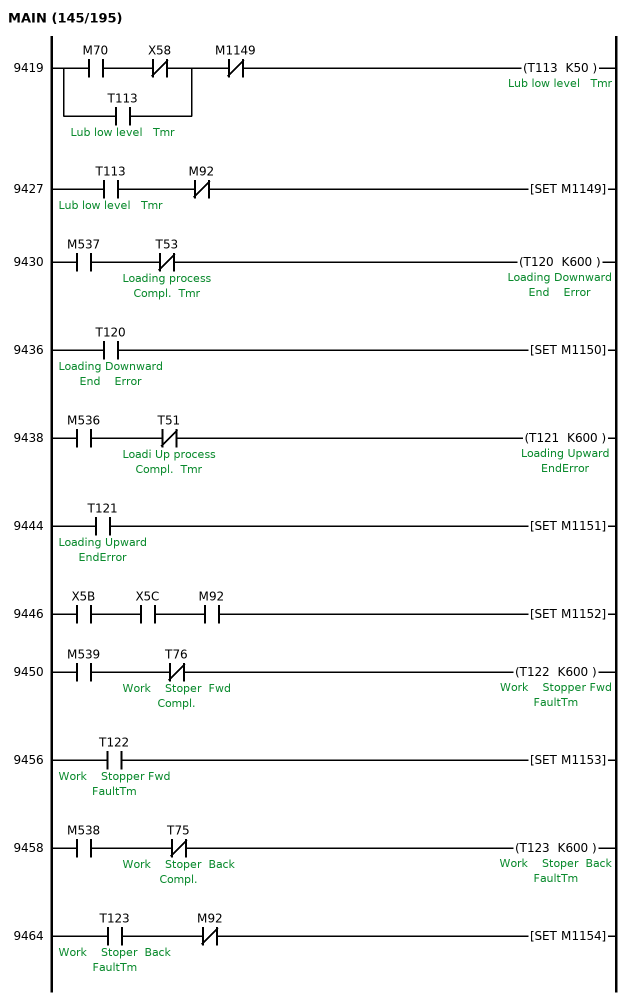
[picture p144: ladder of MAIN, rungs at steps 9419 to 9464]
9419  LD      M70
      ANI     X58
      OR      T113  ; Lub low level   Tmr
      ANI     M1149
      OUT     T113 K50  ; Lub low level   Tmr
9427  LD      T113  ; Lub low level   Tmr
      ANI     M92
      SET     M1149
9430  LD      M537
      ANI     T53  ; Loading process Compl.  Tmr
      OUT     T120 K600  ; Loading Downward End    Error
9436  LD      T120  ; Loading Downward End    Error
      SET     M1150
9438  LD      M536
      ANI     T51  ; Loadi Up process Compl.  Tmr
      OUT     T121 K600  ; Loading Upward  EndError
9444  LD      T121  ; Loading Upward  EndError
      SET     M1151
9446  LD      X5B
      AND     X5C
      AND     M92
      SET     M1152
9450  LD      M539
      ANI     T76  ; Work    Stoper  Fwd     Compl.
      OUT     T122 K600  ; Work    Stopper Fwd     FaultTm
9456  LD      T122  ; Work    Stopper Fwd     FaultTm
      SET     M1153
9458  LD      M538
      ANI     T75  ; Work    Stoper  Back    Compl.
      OUT     T123 K600  ; Work    Stoper  Back    FaultTm
9464  LD      T123  ; Work    Stoper  Back    FaultTm
      ANI     M92
      SET     M1154
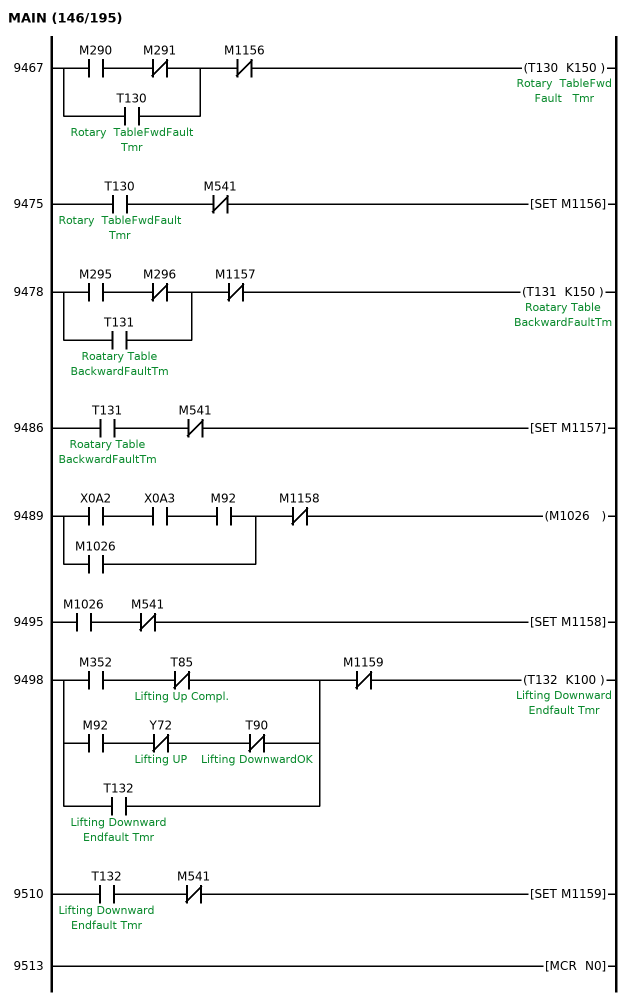
9467  LD      M290
      ANI     M291
      OR      T130  ; Rotary  TableFwdFault   Tmr
      ANI     M1156
      OUT     T130 K150  ; Rotary  TableFwdFault   Tmr
9475  LD      T130  ; Rotary  TableFwdFault   Tmr
      ANI     M541
      SET     M1156
9478  LD      M295
      ANI     M296
      OR      T131  ; Roatary Table   BackwardFaultTm
      ANI     M1157
      OUT     T131 K150  ; Roatary Table   BackwardFaultTm
9486  LD      T131  ; Roatary Table   BackwardFaultTm
      ANI     M541
      SET     M1157
9489  LD      X0A2
      AND     X0A3
      AND     M92
      OR      M1026
      ANI     M1158
      OUT     M1026
9495  LD      M1026
      ANI     M541
      SET     M1158
9498  LD      M352
      ANI     T85  ; Lifting Up Compl.
      LD      M92
      ANI     Y72  ; Lifting UP
      ANI     T90  ; Lifting DownwardOK
      ORB
      OR      T132  ; Lifting DownwardEndfault Tmr
      ANI     M1159
      OUT     T132 K100  ; Lifting DownwardEndfault Tmr
9510  LD      T132  ; Lifting DownwardEndfault Tmr
      ANI     M541
      SET     M1159
9513  MCR     N0
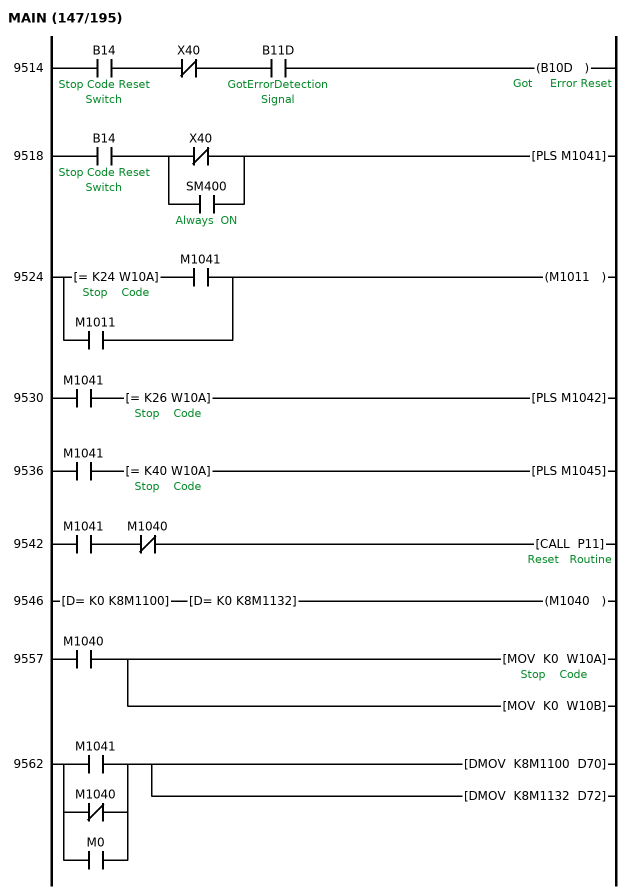
9514  LD      B14  ; Stop Code Reset Switch
      ANI     X40
      AND     B11D  ; GotErrorDetection Signal
      OUT     B10D  ; Got     Error Reset
9518  LD      B14  ; Stop Code Reset Switch
      LDI     X40
      OR      SM400  ; Always  ON
      ANB
      PLS     M1041
9524  LD=     K24 W10A  ; Stop    Code
      AND     M1041
      OR      M1011
      OUT     M1011
9530  LD      M1041
      AND=    K26 W10A  ; Stop    Code
      PLS     M1042
9536  LD      M1041
      AND=    K40 W10A  ; Stop    Code
      PLS     M1045
9542  LD      M1041
      ANI     M1040
      CALL    P11  ; Reset   Routine
9546  LDD=    K0 K8M1100
      ANDD=   K0 K8M1132
      OUT     M1040
9557  LD      M1040
      MOV     K0 W10A
      MOV     K0 W10B
9562  LD      M1041
      ORI     M1040
      OR      M0
      DMOV    K8M1100 D70
      DMOV    K8M1132 D72
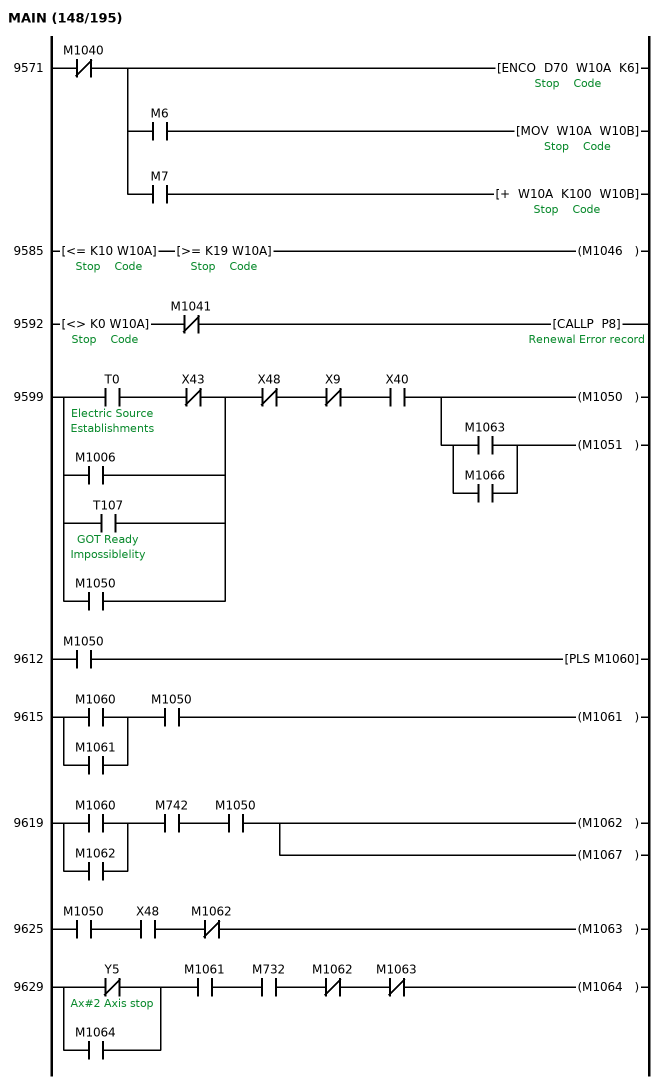
9571  LDI     M1040
      ENCO    D70 W10A K6
      MPS
      AND     M6
      MOV     W10A W10B
      MPP
      AND     M7
      +       W10A K100 W10B
9585  LD<=    K10 W10A  ; Stop    Code
      AND>=   K19 W10A  ; Stop    Code
      OUT     M1046
9592  LD<>    K0 W10A  ; Stop    Code
      ANI     M1041
      CALLP   P8  ; Renewal Error record
9599  LD      T0  ; Electric Source Establishments
      ANI     X43
      OR      M1006
      OR      T107  ; GOT Ready Impossiblelity
      OR      M1050
      ANI     X48
      ANI     X9
      AND     X40
      OUT     M1050
      LD      M1063
      OR      M1066
      ANB
      OUT     M1051
9612  LD      M1050
      PLS     M1060
9615  LD      M1060
      OR      M1061
      AND     M1050
      OUT     M1061
9619  LD      M1060
      OR      M1062
      AND     M742
      AND     M1050
      OUT     M1062
      OUT     M1067
9625  LD      M1050
      AND     X48
      ANI     M1062
      OUT     M1063
9629  LDI     Y5  ; Ax#2 Axis stop
      OR      M1064
      AND     M1061
      AND     M732
      ANI     M1062
      ANI     M1063
      OUT     M1064
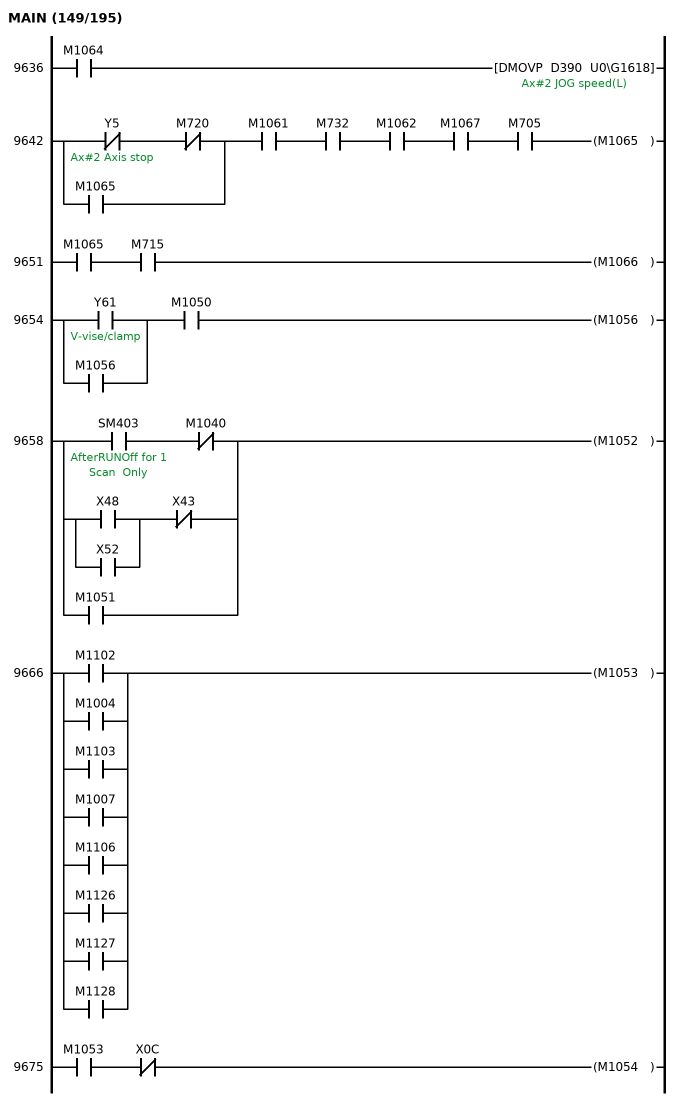
9636  LD      M1064
      DMOVP   D390 U0\G1618
9642  LDI     Y5  ; Ax#2 Axis stop
      ANI     M720
      OR      M1065
      AND     M1061
      AND     M732
      AND     M1062
      AND     M1067
      AND     M705
      OUT     M1065
9651  LD      M1065
      AND     M715
      OUT     M1066
9654  LD      Y61  ; V-vise/clamp
      OR      M1056
      AND     M1050
      OUT     M1056
9658  LD      SM403  ; AfterRUNOff for 1 Scan  Only
      ANI     M1040
      LD      X48
      OR      X52
      ANI     X43
      ORB
      OR      M1051
      OUT     M1052
9666  LD      M1102
      OR      M1004
      OR      M1103
      OR      M1007
      OR      M1106
      OR      M1126
      OR      M1127
      OR      M1128
      OUT     M1053
9675  LD      M1053
      ANI     X0C
      OUT     M1054
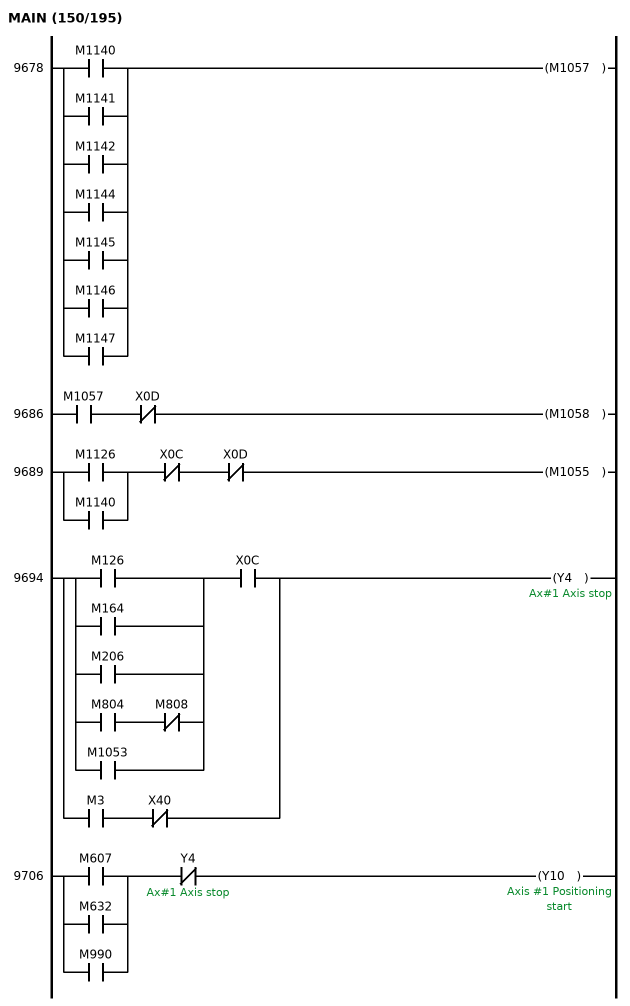
9678  LD      M1140
      OR      M1141
      OR      M1142
      OR      M1144
      OR      M1145
      OR      M1146
      OR      M1147
      OUT     M1057
9686  LD      M1057
      ANI     X0D
      OUT     M1058
9689  LD      M1126
      OR      M1140
      ANI     X0C
      ANI     X0D
      OUT     M1055
9694  LD      M126
      OR      M164
      OR      M206
      LD      M804
      ANI     M808
      ORB
      OR      M1053
      AND     X0C
      LD      M3
      ANI     X40
      ORB
      OUT     Y4  ; Ax#1 Axis stop
9706  LD      M607
      OR      M632
      OR      M990
      ANI     Y4  ; Ax#1 Axis stop
      OUT     Y10  ; Axis #1 Positioning start
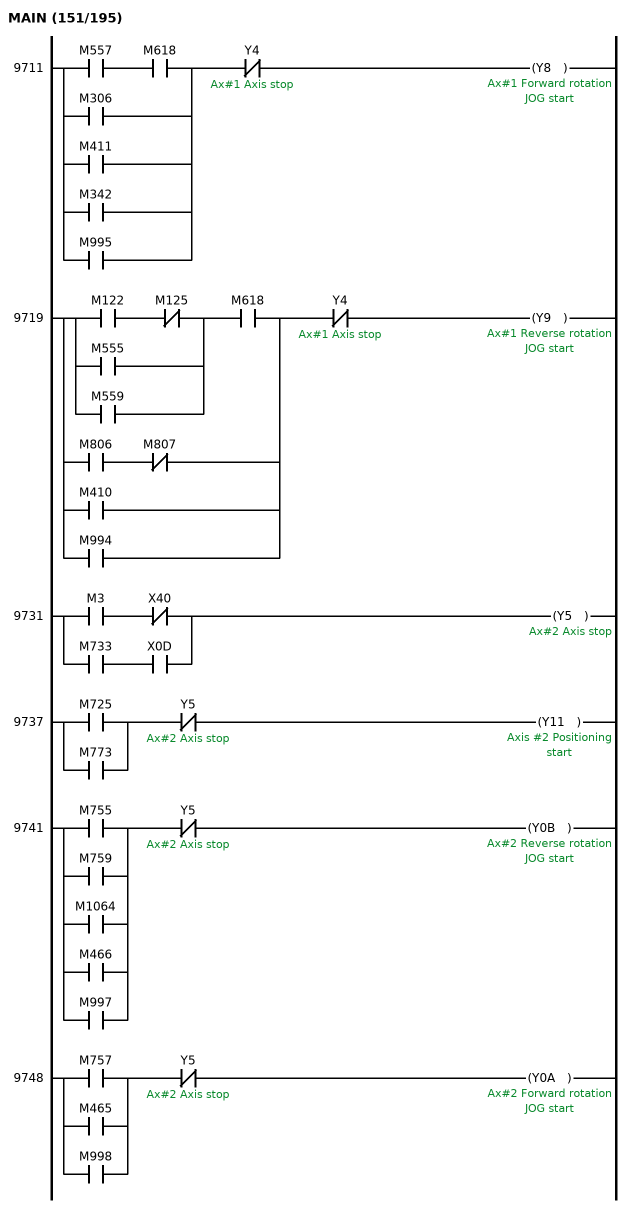
9711  LD      M557
      AND     M618
      OR      M306
      OR      M411
      OR      M342
      OR      M995
      ANI     Y4  ; Ax#1 Axis stop
      OUT     Y8  ; Ax#1 Forward rotation JOG start
9719  LD      M122
      ANI     M125
      OR      M555
      OR      M559
      AND     M618
      LD      M806
      ANI     M807
      ORB
      OR      M410
      OR      M994
      ANI     Y4  ; Ax#1 Axis stop
      OUT     Y9  ; Ax#1 Reverse rotation JOG start
9731  LD      M3
      ANI     X40
      LD      M733
      AND     X0D
      ORB
      OUT     Y5  ; Ax#2 Axis stop
9737  LD      M725
      OR      M773
      ANI     Y5  ; Ax#2 Axis stop
      OUT     Y11  ; Axis #2 Positioning start
9741  LD      M755
      OR      M759
      OR      M1064
      OR      M466
      OR      M997
      ANI     Y5  ; Ax#2 Axis stop
      OUT     Y0B  ; Ax#2 Reverse rotation JOG start
9748  LD      M757
      OR      M465
      OR      M998
      ANI     Y5  ; Ax#2 Axis stop
      OUT     Y0A  ; Ax#2 Forward rotation JOG start
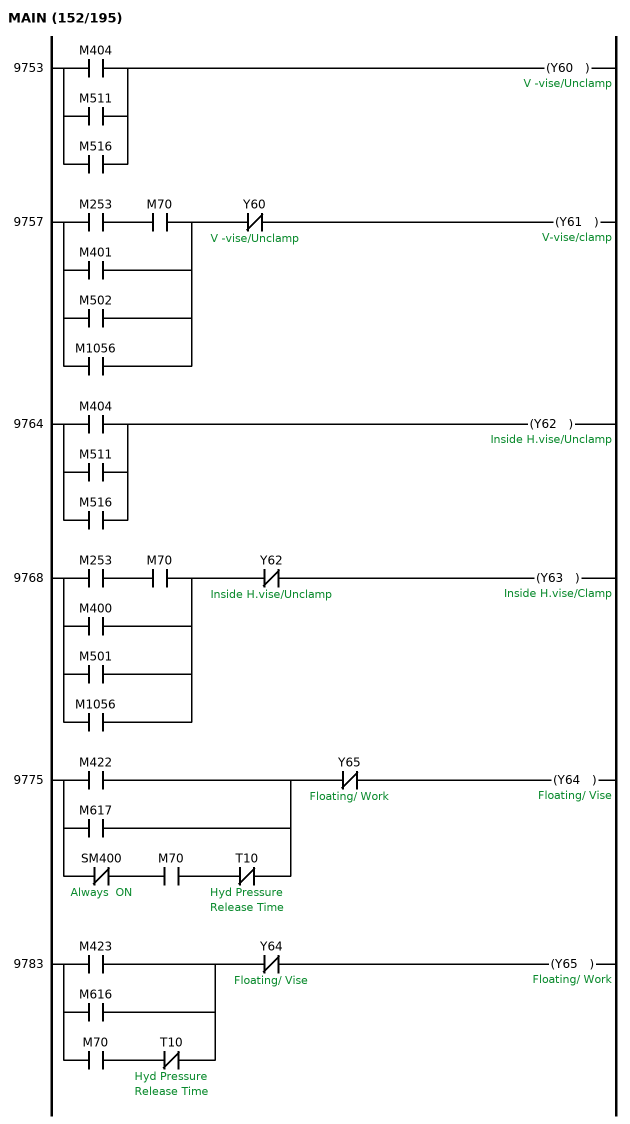
9753  LD      M404
      OR      M511
      OR      M516
      OUT     Y60  ; V -vise/Unclamp
9757  LD      M253
      AND     M70
      OR      M401
      OR      M502
      OR      M1056
      ANI     Y60  ; V -vise/Unclamp
      OUT     Y61  ; V-vise/clamp
9764  LD      M404
      OR      M511
      OR      M516
      OUT     Y62  ; Inside H.vise/Unclamp
9768  LD      M253
      AND     M70
      OR      M400
      OR      M501
      OR      M1056
      ANI     Y62  ; Inside H.vise/Unclamp
      OUT     Y63  ; Inside H.vise/Clamp
9775  LD      M422
      OR      M617
      LDI     SM400  ; Always  ON
      AND     M70
      ANI     T10  ; Hyd Pressure    Release Time
      ORB
      ANI     Y65  ; Floating/ Work
      OUT     Y64  ; Floating/ Vise
9783  LD      M423
      OR      M616
      LD      M70
      ANI     T10  ; Hyd Pressure    Release Time
      ORB
      ANI     Y64  ; Floating/ Vise
      OUT     Y65  ; Floating/ Work
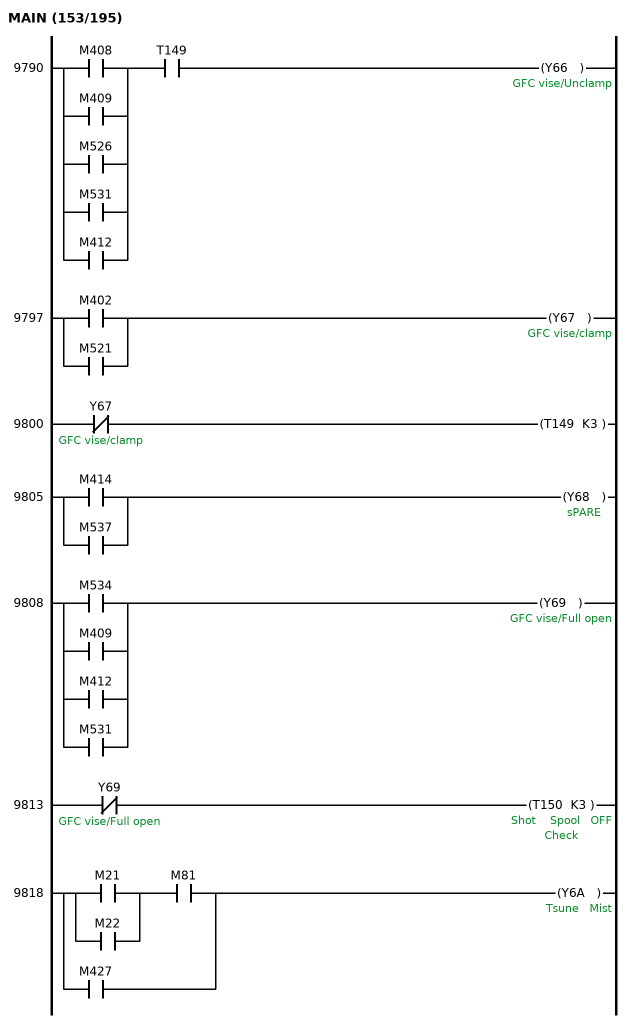
9790  LD      M408
      OR      M409
      OR      M526
      OR      M531
      OR      M412
      AND     T149
      OUT     Y66  ; GFC vise/Unclamp
9797  LD      M402
      OR      M521
      OUT     Y67  ; GFC vise/clamp
9800  LDI     Y67  ; GFC vise/clamp
      OUT     T149 K3
9805  LD      M414
      OR      M537
      OUT     Y68  ; sPARE
9808  LD      M534
      OR      M409
      OR      M412
      OR      M531
      OUT     Y69  ; GFC vise/Full open
9813  LDI     Y69  ; GFC vise/Full open
      OUT     T150 K3  ; Shot    Spool   OFF     Check
9818  LD      M21
      OR      M22
      AND     M81
      OR      M427
      OUT     Y6A  ; Tsune   Mist
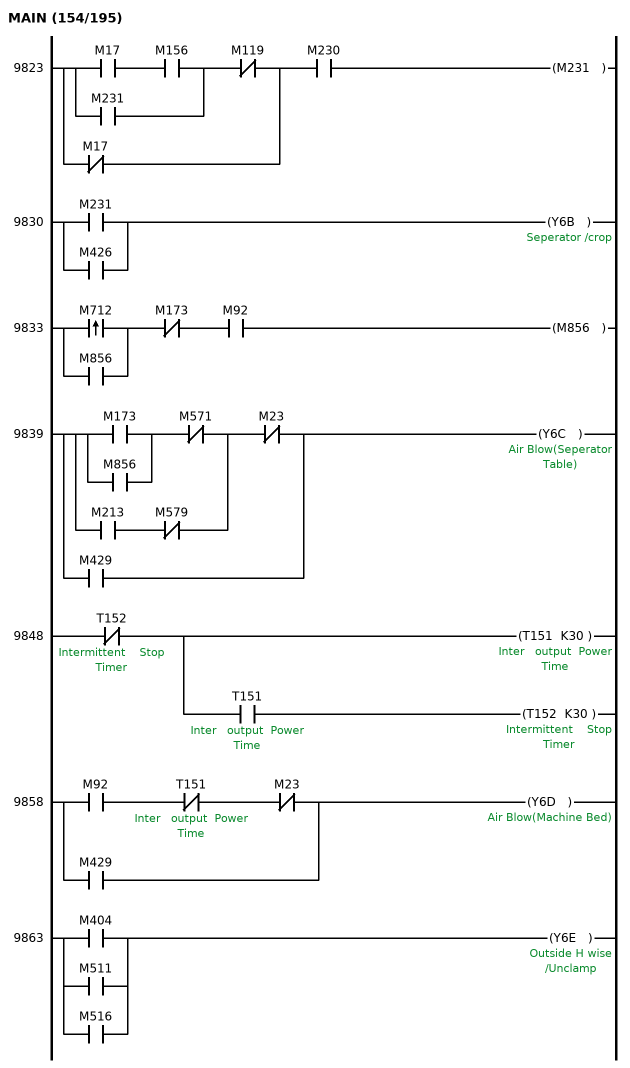
9823  LD      M17
      AND     M156
      OR      M231
      ANI     M119
      ORI     M17
      AND     M230
      OUT     M231
9830  LD      M231
      OR      M426
      OUT     Y6B  ; Seperator /crop
9833  LDP     M712
      OR      M856
      ANI     M173
      AND     M92
      OUT     M856
9839  LD      M173
      OR      M856
      ANI     M571
      LD      M213
      ANI     M579
      ORB
      ANI     M23
      OR      M429
      OUT     Y6C  ; Air Blow(Seperator Table)
9848  LDI     T152  ; Intermittent    Stop    Timer
      OUT     T151 K30  ; Inter   output  Power   Time
      AND     T151  ; Inter   output  Power   Time
      OUT     T152 K30  ; Intermittent    Stop    Timer
9858  LD      M92
      ANI     T151  ; Inter   output  Power   Time
      ANI     M23
      OR      M429
      OUT     Y6D  ; Air Blow(Machine Bed)
9863  LD      M404
      OR      M511
      OR      M516
      OUT     Y6E  ; Outside H wise /Unclamp
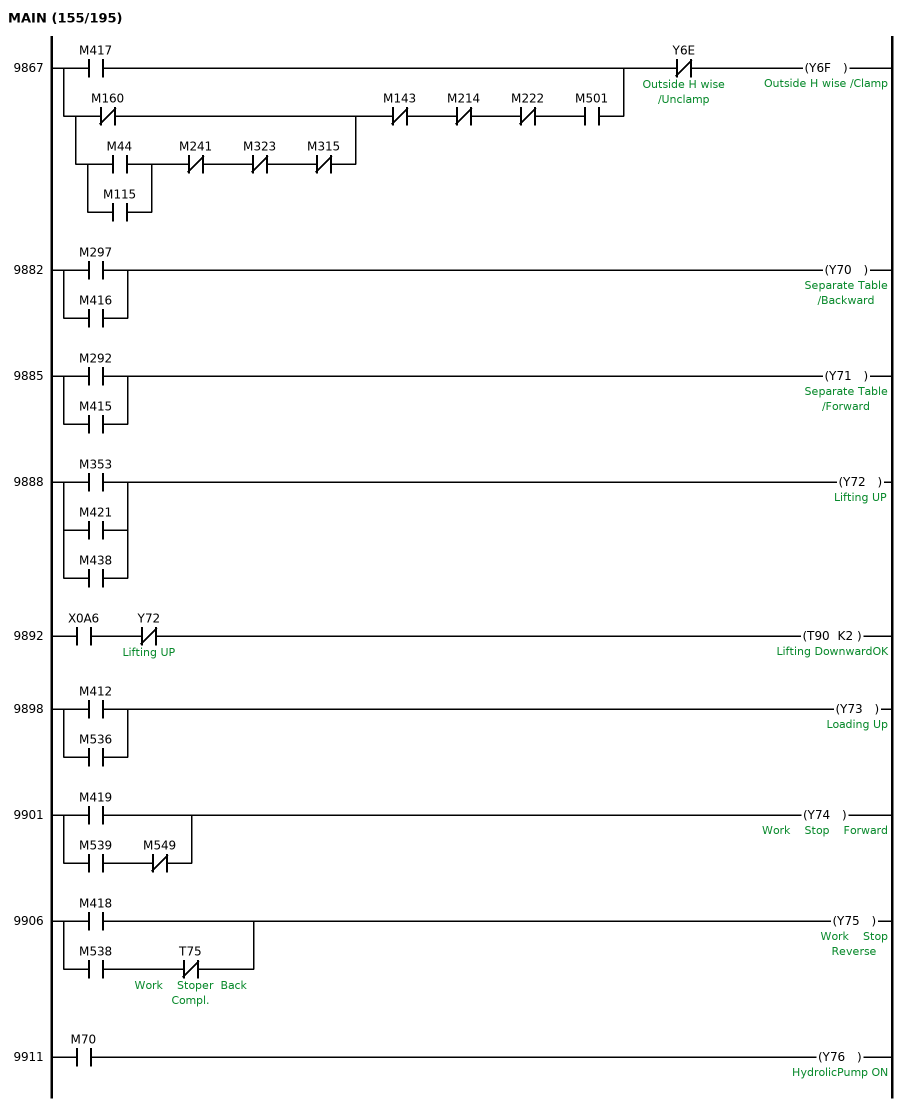
9867  LD      M417
      LDI     M160
      LD      M44
      OR      M115
      ANI     M241
      ANI     M323
      ANI     M315
      ORB
      ANI     M143
      ANI     M214
      ANI     M222
      AND     M501
      ORB
      ANI     Y6E  ; Outside H wise /Unclamp
      OUT     Y6F  ; Outside H wise /Clamp
9882  LD      M297
      OR      M416
      OUT     Y70  ; Separate Table /Backward
9885  LD      M292
      OR      M415
      OUT     Y71  ; Separate Table /Forward
9888  LD      M353
      OR      M421
      OR      M438
      OUT     Y72  ; Lifting UP
9892  LD      X0A6
      ANI     Y72  ; Lifting UP
      OUT     T90 K2  ; Lifting DownwardOK
9898  LD      M412
      OR      M536
      OUT     Y73  ; Loading Up
9901  LD      M419
      LD      M539
      ANI     M549
      ORB
      OUT     Y74  ; Work    Stop    Forward
9906  LD      M418
      LD      M538
      ANI     T75  ; Work    Stoper  Back    Compl.
      ORB
      OUT     Y75  ; Work    Stop    Reverse
9911  LD      M70
      OUT     Y76  ; HydrolicPump ON
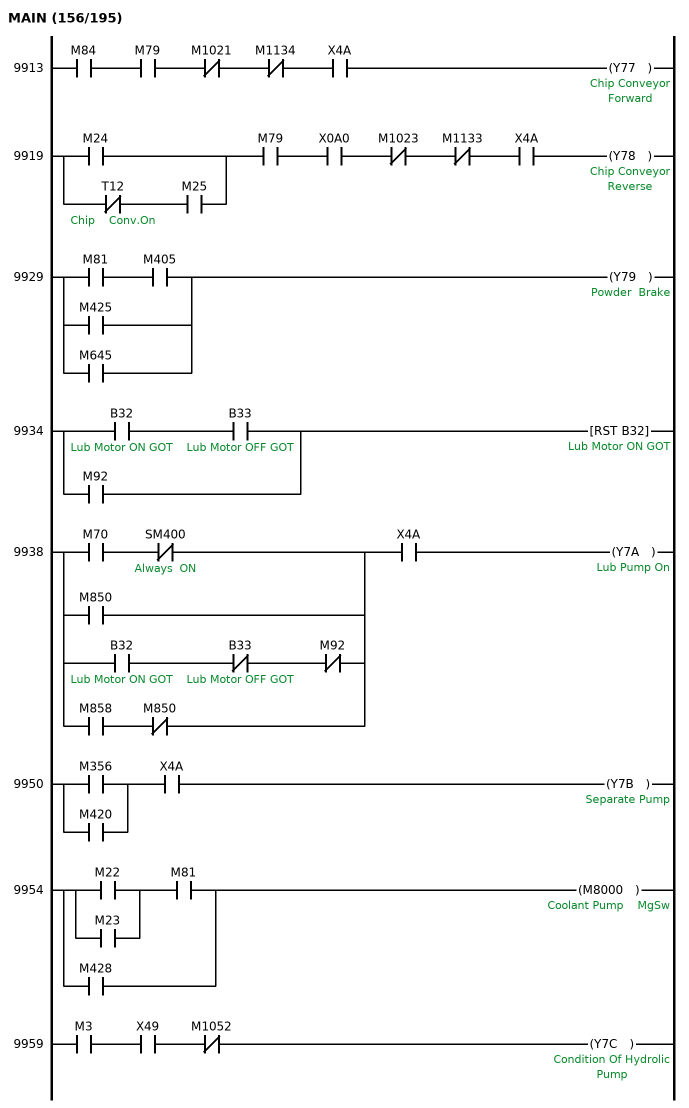
9913  LD      M84
      AND     M79
      ANI     M1021
      ANI     M1134
      AND     X4A
      OUT     Y77  ; Chip Conveyor Forward
9919  LD      M24
      LDI     T12  ; Chip    Conv.On
      AND     M25
      ORB
      AND     M79
      AND     X0A0
      ANI     M1023
      ANI     M1133
      AND     X4A
      OUT     Y78  ; Chip Conveyor Reverse
9929  LD      M81
      AND     M405
      OR      M425
      OR      M645
      OUT     Y79  ; Powder  Brake
9934  LD      B32  ; Lub Motor ON GOT
      AND     B33  ; Lub Motor OFF GOT
      OR      M92
      RST     B32  ; Lub Motor ON GOT
9938  LD      M70
      ANI     SM400  ; Always  ON
      OR      M850
      LD      B32  ; Lub Motor ON GOT
      ANI     B33  ; Lub Motor OFF GOT
      ANI     M92
      ORB
      LD      M858
      ANI     M850
      ORB
      AND     X4A
      OUT     Y7A  ; Lub Pump On
9950  LD      M356
      OR      M420
      AND     X4A
      OUT     Y7B  ; Separate Pump
9954  LD      M22
      OR      M23
      AND     M81
      OR      M428
      OUT     M8000  ; Coolant Pump    MgSw
9959  LD      M3
      AND     X49
      ANI     M1052
      OUT     Y7C  ; Condition Of Hydrolic Pump
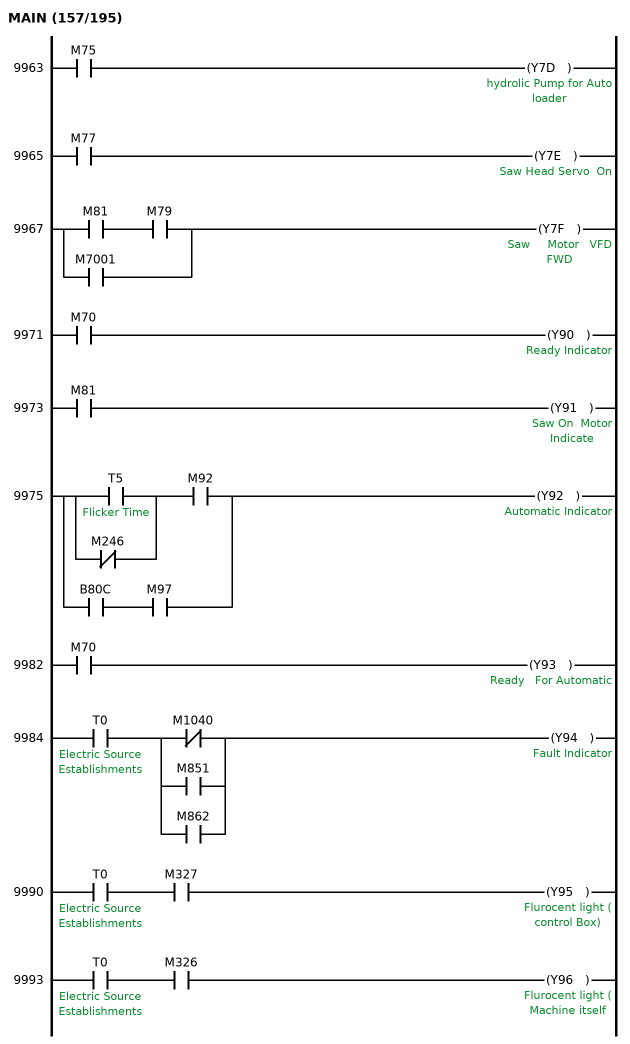
9963  LD      M75
      OUT     Y7D  ; hydrolic Pump for Auto loader
9965  LD      M77
      OUT     Y7E  ; Saw Head Servo  On
9967  LD      M81
      AND     M79
      OR      M7001
      OUT     Y7F  ; Saw     Motor   VFD FWD
9971  LD      M70
      OUT     Y90  ; Ready Indicator
9973  LD      M81
      OUT     Y91  ; Saw On  Motor   Indicate
9975  LD      T5  ; Flicker Time
      ORI     M246
      AND     M92
      LD      B80C
      AND     M97
      ORB
      OUT     Y92  ; Automatic Indicator
9982  LD      M70
      OUT     Y93  ; Ready   For Automatic
9984  LD      T0  ; Electric Source Establishments
      LDI     M1040
      OR      M851
      OR      M862
      ANB
      OUT     Y94  ; Fault Indicator
9990  LD      T0  ; Electric Source Establishments
      AND     M327
      OUT     Y95  ; Flurocent light ( control Box)
9993  LD      T0  ; Electric Source Establishments
      AND     M326
      OUT     Y96  ; Flurocent light ( Machine itself
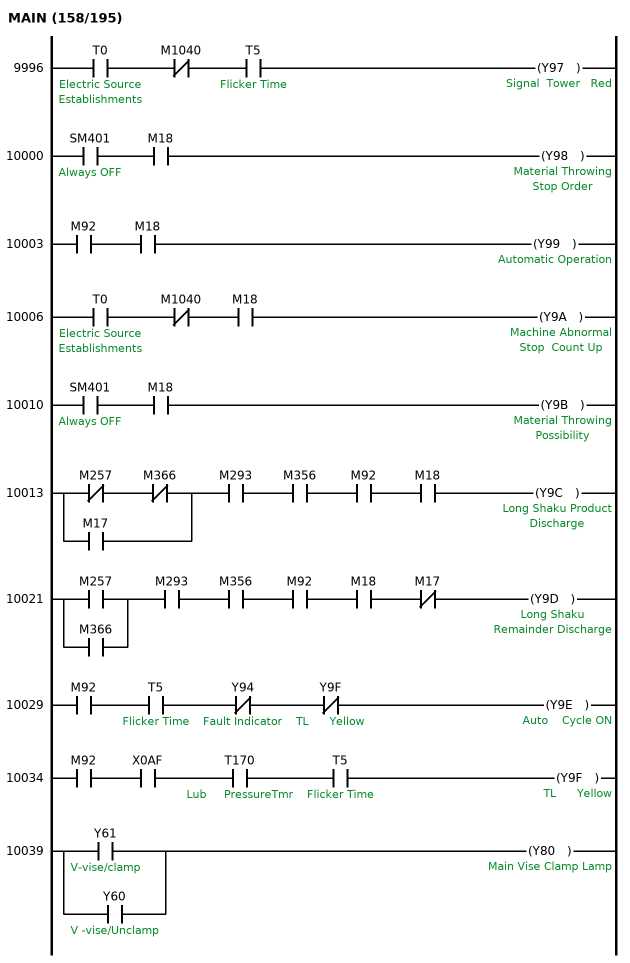
9996  LD      T0  ; Electric Source Establishments
      ANI     M1040
      AND     T5  ; Flicker Time
      OUT     Y97  ; Signal  Tower   Red
10000 LD      SM401  ; Always OFF
      AND     M18
      OUT     Y98  ; Material Throwing Stop Order
10003 LD      M92
      AND     M18
      OUT     Y99  ; Automatic Operation
10006 LD      T0  ; Electric Source Establishments
      ANI     M1040
      AND     M18
      OUT     Y9A  ; Machine Abnormal Stop  Count Up
10010 LD      SM401  ; Always OFF
      AND     M18
      OUT     Y9B  ; Material Throwing Possibility
10013 LDI     M257
      ANI     M366
      OR      M17
      AND     M293
      AND     M356
      AND     M92
      AND     M18
      OUT     Y9C  ; Long Shaku Product Discharge
10021 LD      M257
      OR      M366
      AND     M293
      AND     M356
      AND     M92
      AND     M18
      ANI     M17
      OUT     Y9D  ; Long Shaku Remainder Discharge
10029 LD      M92
      AND     T5  ; Flicker Time
      ANI     Y94  ; Fault Indicator
      ANI     Y9F  ; TL      Yellow
      OUT     Y9E  ; Auto    Cycle ON
10034 LD      M92
      AND     X0AF
      AND     T170  ; Lub     PressureTmr
      AND     T5  ; Flicker Time
      OUT     Y9F  ; TL      Yellow
10039 LD      Y61  ; V-vise/clamp
      OR      Y60  ; V -vise/Unclamp
      OUT     Y80  ; Main Vise Clamp Lamp
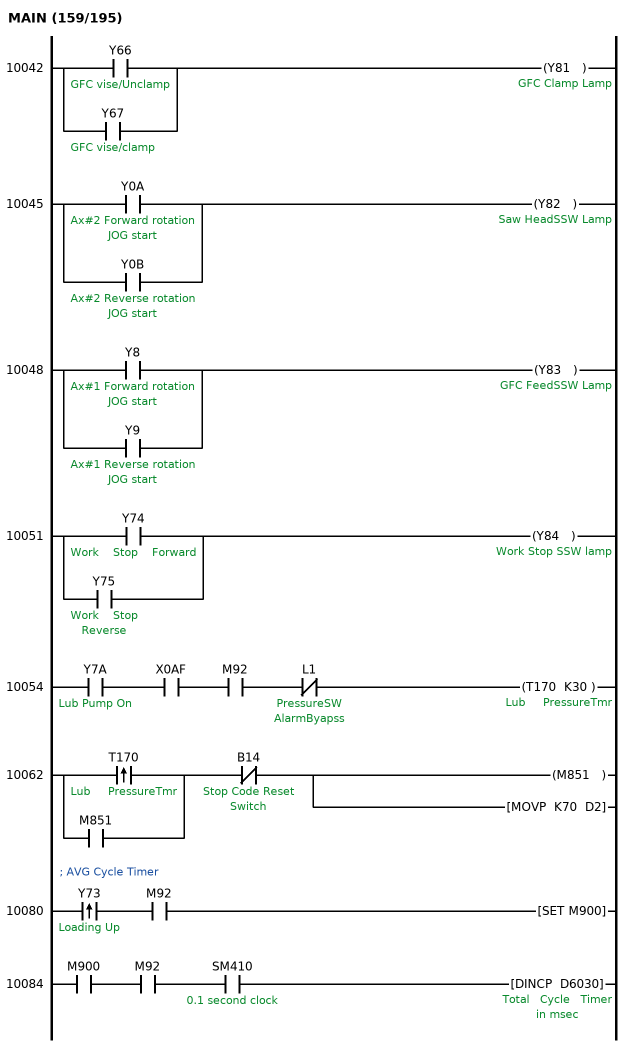
10042 LD      Y66  ; GFC vise/Unclamp
      OR      Y67  ; GFC vise/clamp
      OUT     Y81  ; GFC Clamp Lamp
10045 LD      Y0A  ; Ax#2 Forward rotation JOG start
      OR      Y0B  ; Ax#2 Reverse rotation JOG start
      OUT     Y82  ; Saw HeadSSW Lamp
10048 LD      Y8  ; Ax#1 Forward rotation JOG start
      OR      Y9  ; Ax#1 Reverse rotation JOG start
      OUT     Y83  ; GFC FeedSSW Lamp
10051 LD      Y74  ; Work    Stop    Forward
      OR      Y75  ; Work    Stop    Reverse
      OUT     Y84  ; Work Stop SSW lamp
10054 LD      Y7A  ; Lub Pump On
      AND     X0AF
      AND     M92
      ANI     L1  ; PressureSW AlarmByapss
      OUT     T170 K30  ; Lub     PressureTmr
10062 LDP     T170  ; Lub     PressureTmr
      OR      M851
      ANI     B14  ; Stop Code Reset Switch
      OUT     M851
      MOVP    K70 D2
; AVG Cycle Timer
10080 LDP     Y73  ; Loading Up
      AND     M92
      SET     M900
10084 LD      M900
      AND     M92
      AND     SM410  ; 0.1 second clock
      DINCP   D6030  ; Total   Cycle   Timer in msec
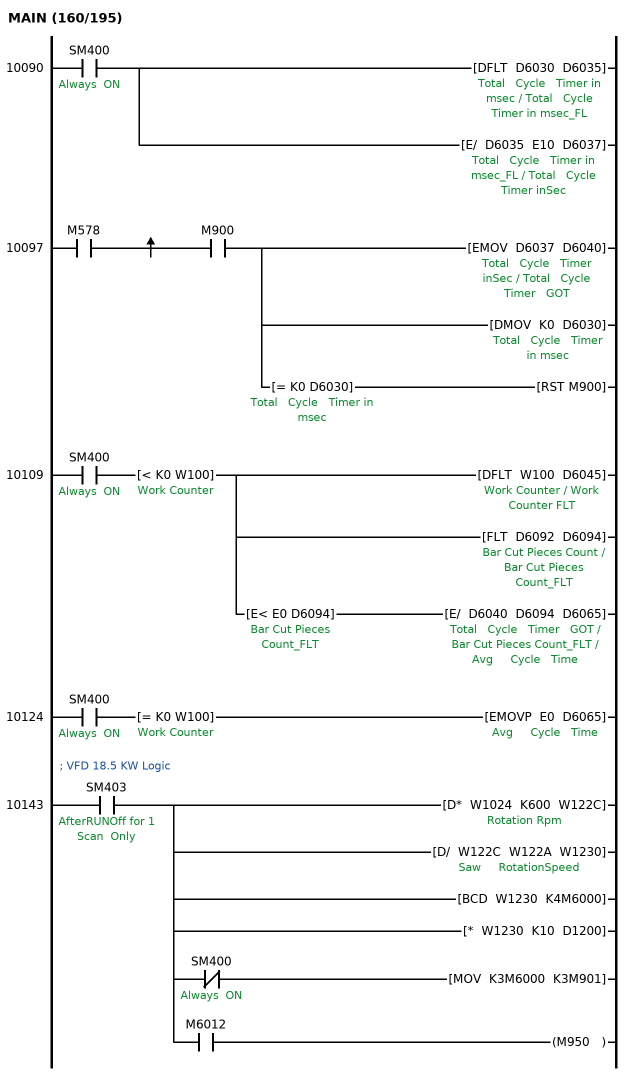
10090 LD      SM400  ; Always  ON
      DFLT    D6030 D6035  ; Total   Cycle   Timer in msec_FL
      E/      D6035 E10 D6037  ; Total   Cycle   Timer inSec
10097 LD      M578
      MEP
      AND     M900
      EMOV    D6037 D6040  ; Total   Cycle   Timer   GOT
      DMOV    K0 D6030
      AND=    K0 D6030  ; Total   Cycle   Timer in msec
      RST     M900
10109 LD      SM400  ; Always  ON
      AND<    K0 W100  ; Work Counter
      DFLT    W100 D6045  ; Work    Counter FLT
      FLT     D6092 D6094  ; Bar Cut Pieces Count_FLT
      ANDE<   E0 D6094  ; Bar Cut Pieces Count_FLT
      E/      D6040 D6094 D6065  ; Avg     Cycle   Time
10124 LD      SM400  ; Always  ON
      AND=    K0 W100  ; Work Counter
      EMOVP   E0 D6065
; VFD 18.5 KW Logic
10143 LD      SM403  ; AfterRUNOff for 1 Scan  Only
      D*      W1024 K600 W122C
      D/      W122C W122A W1230  ; Saw     RotationSpeed
      BCD     W1230 K4M6000
      *       W1230 K10 D1200
      MPS
      ANI     SM400  ; Always  ON
      MOV     K3M6000 K3M901
      MPP
      AND     M6012
      OUT     M950
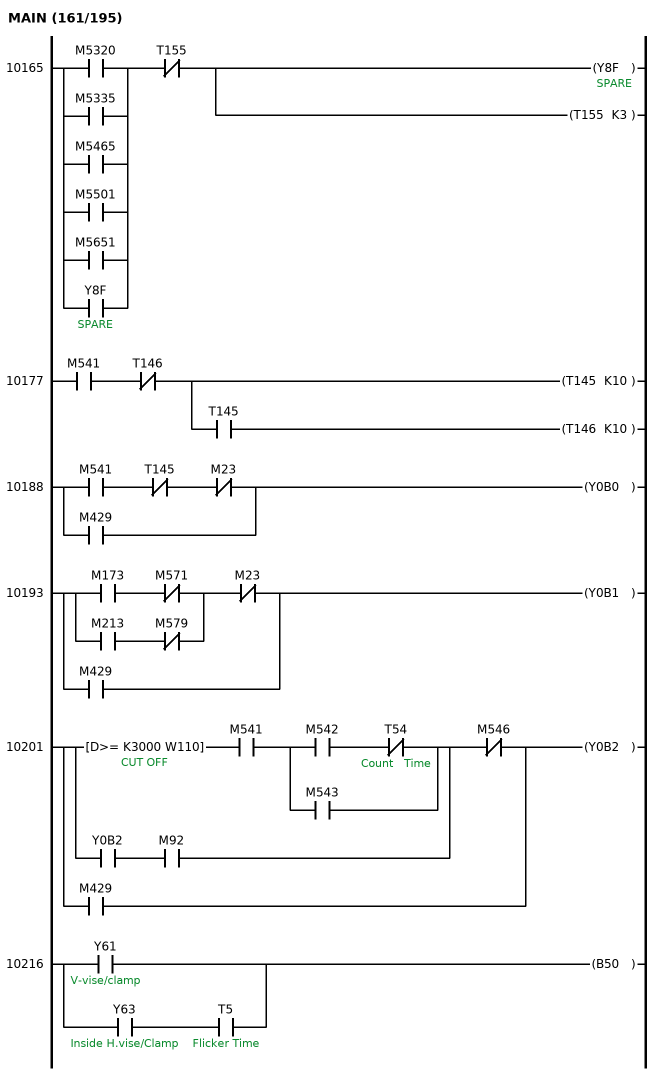
10165 LD      M5320
      OR      M5335
      OR      M5465
      OR      M5501
      OR      M5651
      OR      Y8F  ; SPARE
      ANI     T155
      OUT     Y8F  ; SPARE
      OUT     T155 K3
10177 LD      M541
      ANI     T146
      OUT     T145 K10
      AND     T145
      OUT     T146 K10
10188 LD      M541
      ANI     T145
      ANI     M23
      OR      M429
      OUT     Y0B0
10193 LD      M173
      ANI     M571
      LD      M213
      ANI     M579
      ORB
      ANI     M23
      OR      M429
      OUT     Y0B1
10201 LDD>=   K3000 W110  ; CUT OFF
      AND     M541
      LD      M542
      ANI     T54  ; Count   Time
      OR      M543
      ANB
      LD      Y0B2
      AND     M92
      ORB
      ANI     M546
      OR      M429
      OUT     Y0B2
10216 LD      Y61  ; V-vise/clamp
      LD      Y63  ; Inside H.vise/Clamp
      AND     T5  ; Flicker Time
      ORB
      OUT     B50
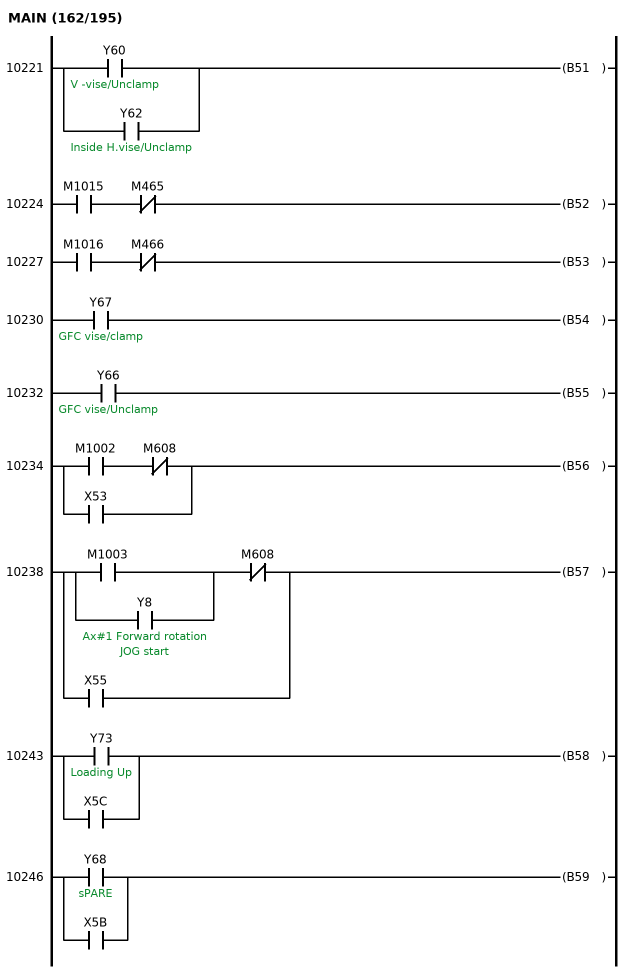
10221 LD      Y60  ; V -vise/Unclamp
      OR      Y62  ; Inside H.vise/Unclamp
      OUT     B51
10224 LD      M1015
      ANI     M465
      OUT     B52
10227 LD      M1016
      ANI     M466
      OUT     B53
10230 LD      Y67  ; GFC vise/clamp
      OUT     B54
10232 LD      Y66  ; GFC vise/Unclamp
      OUT     B55
10234 LD      M1002
      ANI     M608
      OR      X53
      OUT     B56
10238 LD      M1003
      OR      Y8  ; Ax#1 Forward rotation JOG start
      ANI     M608
      OR      X55
      OUT     B57
10243 LD      Y73  ; Loading Up
      OR      X5C
      OUT     B58
10246 LD      Y68  ; sPARE
      OR      X5B
      OUT     B59
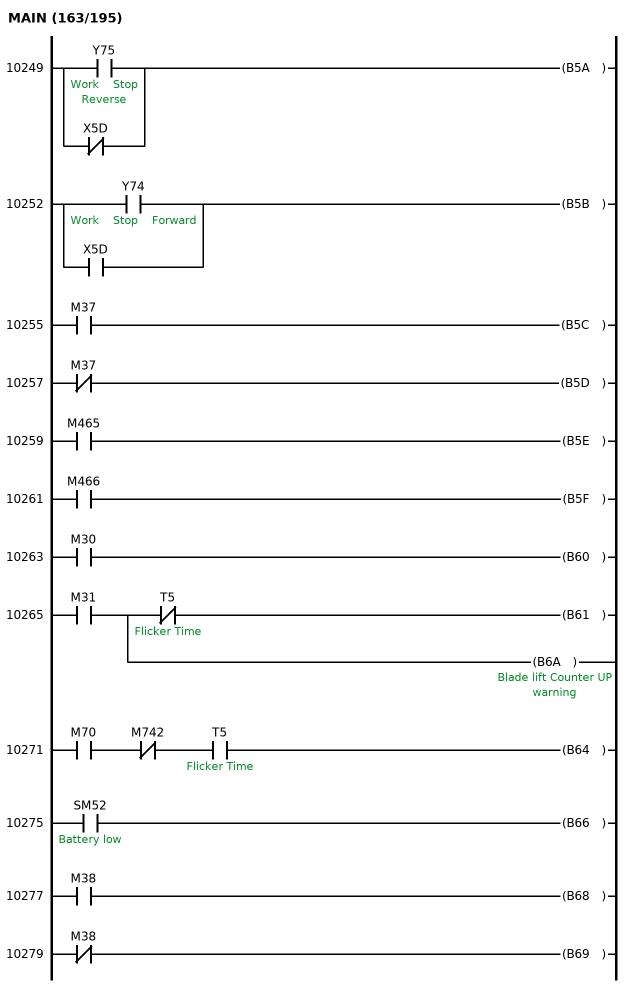
10249 LD      Y75  ; Work    Stop    Reverse
      ORI     X5D
      OUT     B5A
10252 LD      Y74  ; Work    Stop    Forward
      OR      X5D
      OUT     B5B
10255 LD      M37
      OUT     B5C
10257 LDI     M37
      OUT     B5D
10259 LD      M465
      OUT     B5E
10261 LD      M466
      OUT     B5F
10263 LD      M30
      OUT     B60
10265 LD      M31
      MPS
      ANI     T5  ; Flicker Time
      OUT     B61
      MPP
      OUT     B6A  ; Blade lift Counter UP warning
10271 LD      M70
      ANI     M742
      AND     T5  ; Flicker Time
      OUT     B64
10275 LD      SM52  ; Battery low
      OUT     B66
10277 LD      M38
      OUT     B68
10279 LDI     M38
      OUT     B69
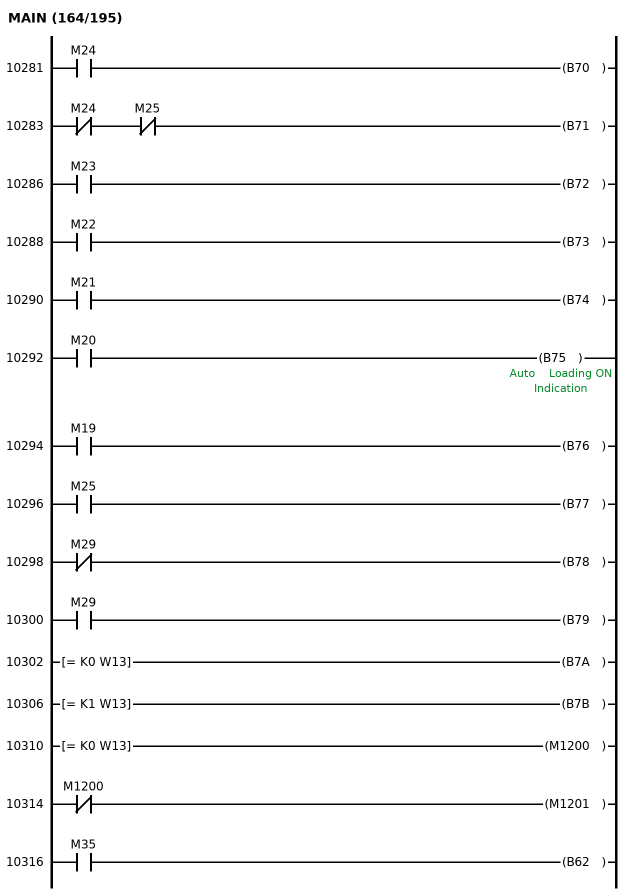
10281 LD      M24
      OUT     B70
10283 LDI     M24
      ANI     M25
      OUT     B71
10286 LD      M23
      OUT     B72
10288 LD      M22
      OUT     B73
10290 LD      M21
      OUT     B74
10292 LD      M20
      OUT     B75  ; Auto    Loading ON Indication
10294 LD      M19
      OUT     B76
10296 LD      M25
      OUT     B77
10298 LDI     M29
      OUT     B78
10300 LD      M29
      OUT     B79
10302 LD=     K0 W13
      OUT     B7A
10306 LD=     K1 W13
      OUT     B7B
10310 LD=     K0 W13
      OUT     M1200
10314 LDI     M1200
      OUT     M1201
10316 LD      M35
      OUT     B62
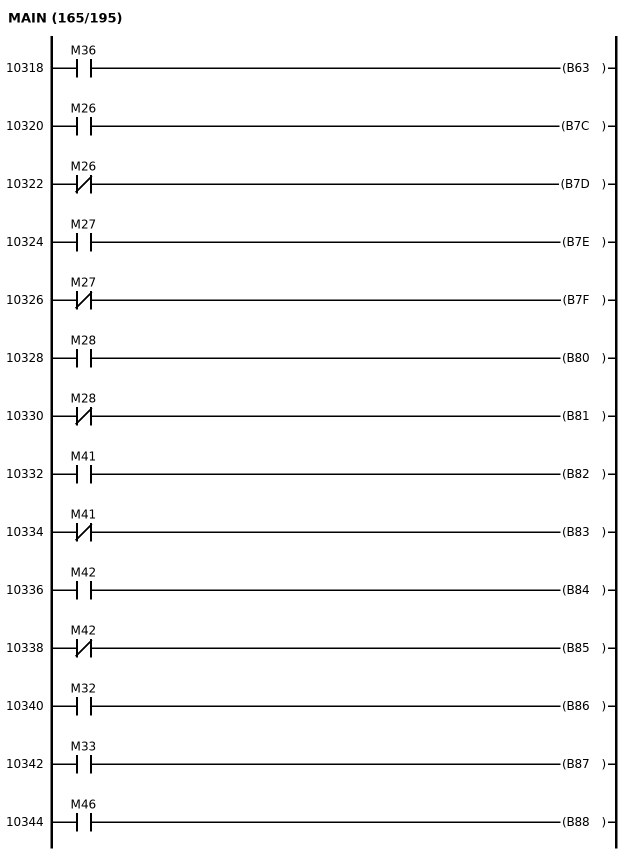
10318 LD      M36
      OUT     B63
10320 LD      M26
      OUT     B7C
10322 LDI     M26
      OUT     B7D
10324 LD      M27
      OUT     B7E
10326 LDI     M27
      OUT     B7F
10328 LD      M28
      OUT     B80
10330 LDI     M28
      OUT     B81
10332 LD      M41
      OUT     B82
10334 LDI     M41
      OUT     B83
10336 LD      M42
      OUT     B84
10338 LDI     M42
      OUT     B85
10340 LD      M32
      OUT     B86
10342 LD      M33
      OUT     B87
10344 LD      M46
      OUT     B88
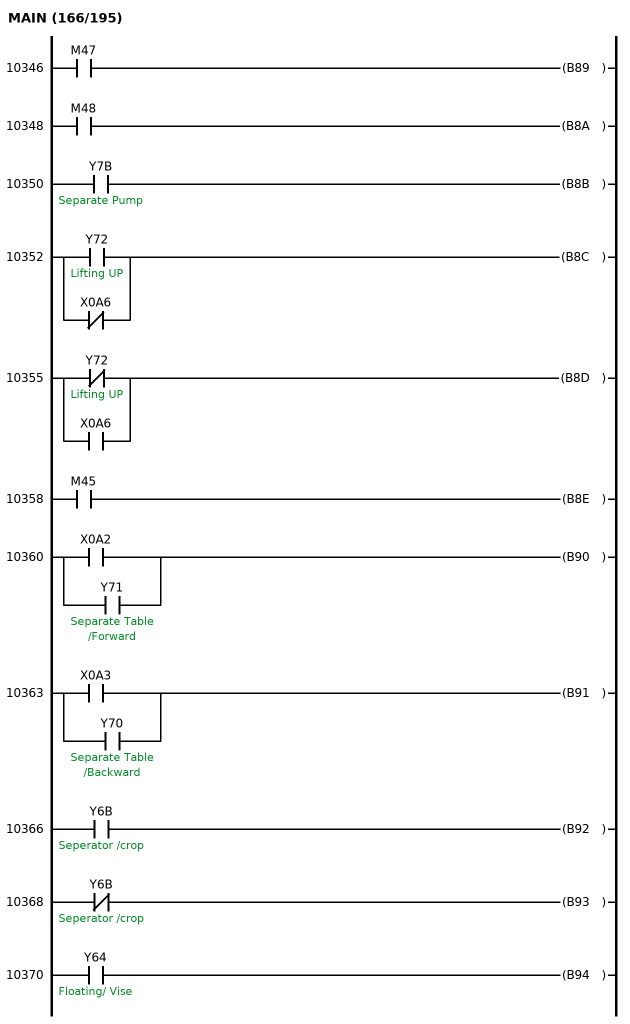
10346 LD      M47
      OUT     B89
10348 LD      M48
      OUT     B8A
10350 LD      Y7B  ; Separate Pump
      OUT     B8B
10352 LD      Y72  ; Lifting UP
      ORI     X0A6
      OUT     B8C
10355 LDI     Y72  ; Lifting UP
      OR      X0A6
      OUT     B8D
10358 LD      M45
      OUT     B8E
10360 LD      X0A2
      OR      Y71  ; Separate Table /Forward
      OUT     B90
10363 LD      X0A3
      OR      Y70  ; Separate Table /Backward
      OUT     B91
10366 LD      Y6B  ; Seperator /crop
      OUT     B92
10368 LDI     Y6B  ; Seperator /crop
      OUT     B93
10370 LD      Y64  ; Floating/ Vise
      OUT     B94
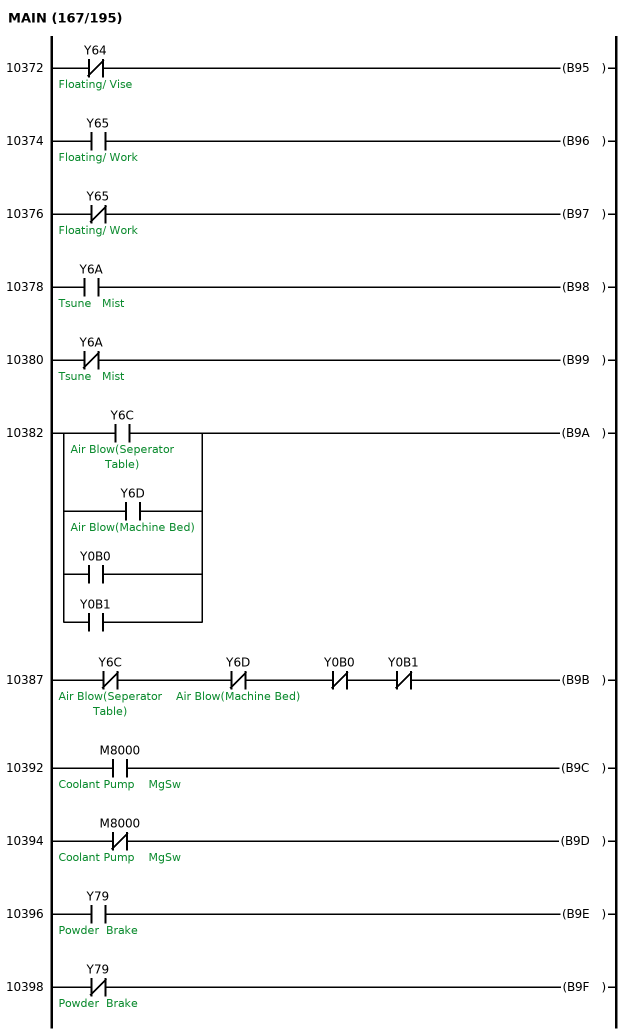
10372 LDI     Y64  ; Floating/ Vise
      OUT     B95
10374 LD      Y65  ; Floating/ Work
      OUT     B96
10376 LDI     Y65  ; Floating/ Work
      OUT     B97
10378 LD      Y6A  ; Tsune   Mist
      OUT     B98
10380 LDI     Y6A  ; Tsune   Mist
      OUT     B99
10382 LD      Y6C  ; Air Blow(Seperator Table)
      OR      Y6D  ; Air Blow(Machine Bed)
      OR      Y0B0
      OR      Y0B1
      OUT     B9A
10387 LDI     Y6C  ; Air Blow(Seperator Table)
      ANI     Y6D  ; Air Blow(Machine Bed)
      ANI     Y0B0
      ANI     Y0B1
      OUT     B9B
10392 LD      M8000  ; Coolant Pump    MgSw
      OUT     B9C
10394 LDI     M8000  ; Coolant Pump    MgSw
      OUT     B9D
10396 LD      Y79  ; Powder  Brake
      OUT     B9E
10398 LDI     Y79  ; Powder  Brake
      OUT     B9F
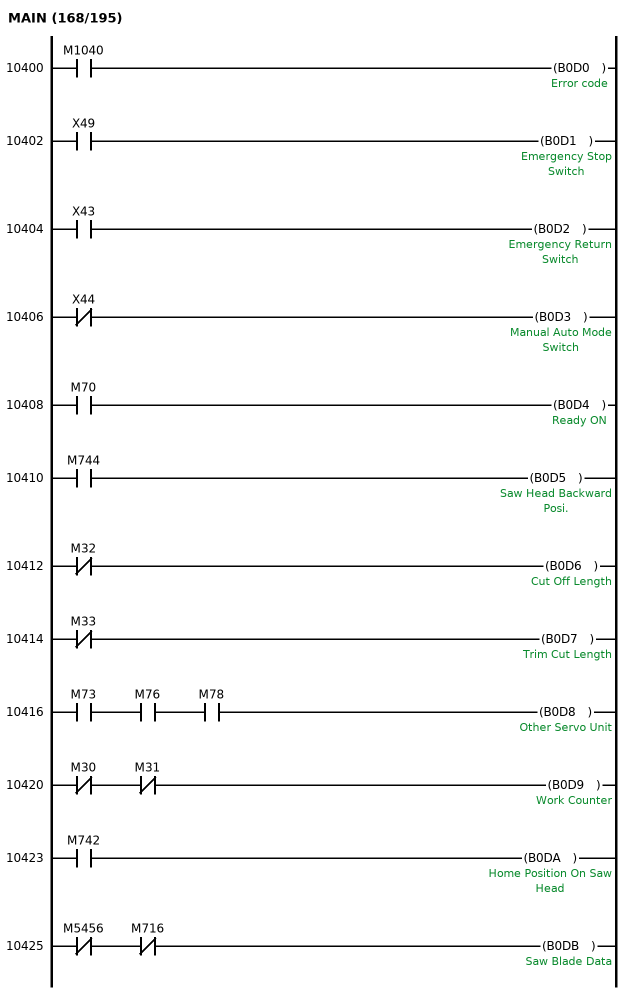
10400 LD      M1040
      OUT     B0D0  ; Error code
10402 LD      X49
      OUT     B0D1  ; Emergency Stop Switch
10404 LD      X43
      OUT     B0D2  ; Emergency Return Switch
10406 LDI     X44
      OUT     B0D3  ; Manual Auto Mode Switch
10408 LD      M70
      OUT     B0D4  ; Ready ON
10410 LD      M744
      OUT     B0D5  ; Saw Head Backward Posi.
10412 LDI     M32
      OUT     B0D6  ; Cut Off Length
10414 LDI     M33
      OUT     B0D7  ; Trim Cut Length
10416 LD      M73
      AND     M76
      AND     M78
      OUT     B0D8  ; Other Servo Unit
10420 LDI     M30
      ANI     M31
      OUT     B0D9  ; Work Counter
10423 LD      M742
      OUT     B0DA  ; Home Position On Saw Head
10425 LDI     M5456
      ANI     M716
      OUT     B0DB  ; Saw Blade Data
